SYSTEM TESTBED_VIEWL (* Testbed View + HMI *)
  (* Standard: 61499 ITA; Classification: Testbed *)
  (* Version 0.3, 2004-10-26, JHC, Rockwell Automation, Changed rotary representation to gate on ring chute. *)
  (* Version 0.2, 2004-10-22, JHC, Rockwell Automation, Reformatted XSPACEs to work with DIA=40 or 25.. *)
  (* Version 0.1, 2004-09-28, JHC, Rockwell Automation, Updated for new conveyor models. *)
  (* Version 0.0, 2002-04-15, JHC, Rockwell Automation *)
  DEVICE HMI : FRAME_DEVICE
    RESOURCE HMI_PANEL : PANEL_RESOURCE
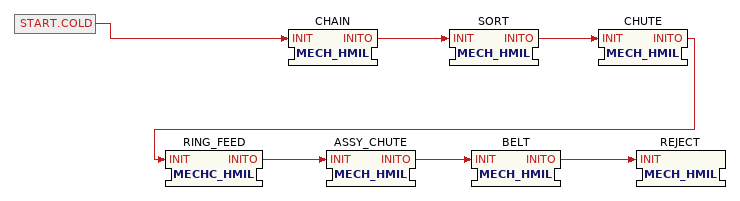
      FBS
        CHAIN : MECH_HMIL;
        SORT : MECH_HMIL;
        CHUTE : MECH_HMIL;
        RING_FEED : MECHC_HMIL;
        ASSY_CHUTE : MECH_HMIL;
        BELT : MECH_HMIL;
        REJECT : MECH_HMIL;
      END_FBS
      EVENT_CONNECTIONS
        START.COLD TO CHAIN.INIT;
        CHAIN.INITO TO SORT.INIT;
        CHUTE.INITO TO RING_FEED.INIT;
        RING_FEED.INITO TO ASSY_CHUTE.INIT;
        SORT.INITO TO CHUTE.INIT;
        BELT.INITO TO REJECT.INIT;
        ASSY_CHUTE.INITO TO BELT.INIT;
      END_CONNECTIONS
    END_RESOURCE
  END_DEVICE
  DEVICE MODEL : FRAME_DEVICE
    RESOURCE CHAIN : VIEW_PANEL
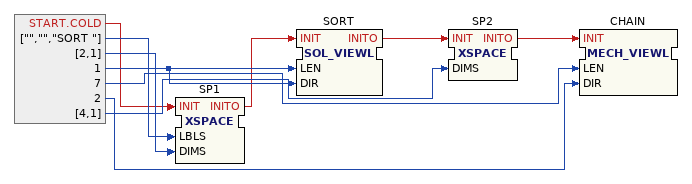
      FBS
        SP1 : XSPACE;
        SORT : SOL_VIEWL; (* Sort Solenoid *)
        SP2 : XSPACE;
        CHAIN : MECH_VIEWL; (* First Chain Segment *)
      END_FBS
      EVENT_CONNECTIONS
        START.COLD TO SP1.INIT;
        SP1.INITO TO SORT.INIT;
        SORT.INITO TO SP2.INIT;
        SP2.INITO TO CHAIN.INIT;
      END_CONNECTIONS
      DATA_CONNECTIONS
        ["","","SORT "] TO SP1.LBLS;
        [2,1] TO SP1.DIMS;
        1 TO SORT.LEN;
        1 TO SORT.DIR;
        7 TO CHAIN.LEN;
        2 TO CHAIN.DIR;
        [4,1] TO SP2.DIMS;
      END_CONNECTIONS
    END_RESOURCE
    RESOURCE CHUTES : VIEW_PANEL
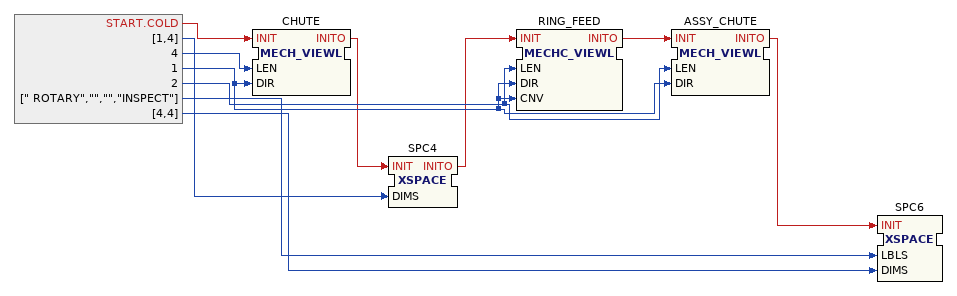
      FBS
        CHUTE : MECH_VIEWL; (* Peg Chute *)
        SPC4 : XSPACE; (* Ring Feed Chute *)
        RING_FEED : MECHC_VIEWL; (* Ring Feed Chute *)
        ASSY_CHUTE : MECH_VIEWL; (* Assembly Chute *)
        SPC6 : XSPACE;
      END_FBS
      EVENT_CONNECTIONS
        START.COLD TO CHUTE.INIT;
        CHUTE.INITO TO SPC4.INIT;
        SPC4.INITO TO RING_FEED.INIT;
        RING_FEED.INITO TO ASSY_CHUTE.INIT;
        ASSY_CHUTE.INITO TO SPC6.INIT;
      END_CONNECTIONS
      DATA_CONNECTIONS
        [1,4] TO SPC4.DIMS;
        4 TO CHUTE.LEN;
        1 TO CHUTE.DIR;
        2 TO RING_FEED.LEN;
        1 TO RING_FEED.DIR;
        2 TO ASSY_CHUTE.LEN;
        1 TO ASSY_CHUTE.DIR;
        [" ROTARY","","","INSPECT"] TO SPC6.LBLS;
        [4,4] TO SPC6.DIMS;
        1 TO RING_FEED.CNV;
      END_CONNECTIONS
    END_RESOURCE
    RESOURCE BELT : VIEW_PANEL
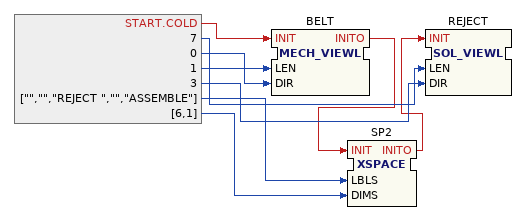
      FBS
        BELT : MECH_VIEWL;
        SP2 : XSPACE;
        REJECT : SOL_VIEWL;
      END_FBS
      EVENT_CONNECTIONS
        START.COLD TO BELT.INIT;
        SP2.INITO TO REJECT.INIT;
        BELT.INITO TO SP2.INIT;
      END_CONNECTIONS
      DATA_CONNECTIONS
        7 TO BELT.LEN;
        0 TO BELT.DIR;
        1 TO REJECT.LEN;
        3 TO REJECT.DIR;
        ["","","REJECT ","","ASSEMBLE"] TO SP2.LBLS;
        [6,1] TO SP2.DIMS;
      END_CONNECTIONS
    END_RESOURCE
    DATA_CONNECTIONS
      40 TO CHUTES.DIA;
      [7,4] TO CHUTES.SIZE;
      1 TO CHUTES.VERTICAL;
      40 TO BELT.DIA;
      [7,2] TO BELT.SIZE;
      0 TO CHAIN.TRACE;
      40 TO CHAIN.DIA;
      [7,2] TO CHAIN.SIZE;
    END_CONNECTIONS
  END_DEVICE
  DATA_CONNECTIONS (* parameter values *)
    [100,100,375,360] TO HMI.BOUNDS;
    [475,100,290,360] TO MODEL.BOUNDS;
    [1,1] TO HMI.GRID;
  END_CONNECTIONS
END_SYSTEM
